TYPE DataFrame EXTENDS SubIndexModuleBase :
STRUCT
END_STRUCT
END_TYPE

(* stored: Version 1.1.0.1, ProductVersion 3.1.4024.3
   DUT DataFrame: Id {24d59139-6f0c-4ba0-8544-3b84c2f40f97} *)
